(* PLC project  *)

CONFIGURATION Empty_Module_20
END_CONFIGURATION
